(* PLC project Senza_nome, Sconosciuto Senza_nome 1 *)
(* stored: creationDateTime 2026-08-27T11:46:05, modificationDateTime 2026-08-27T11:49:45 *)

PROGRAM program0
  VAR
    S1 : BOOL;
    LED : BOOL;
  END_VAR

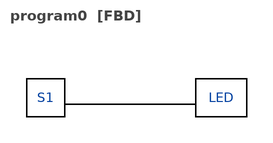
(* FBD diagram, written out as Structured Text *)
LED := S1;
END_PROGRAM

CONFIGURATION Config0
  RESOURCE Res0 ON PLC
    TASK task0(INTERVAL := T#20ms, PRIORITY := 0);
    PROGRAM instance0 WITH task0 : program0;
  END_RESOURCE
END_CONFIGURATION
